(* PLC project  *)

CONFIGURATION StepIM_Extra
END_CONFIGURATION
